// TwinCAT 3 PLC project GettingStarted
// ProgramVersion: 3.1.4026.20
// libraries:
//   Tc2_Standard, * (Beckhoff Automation GmbH)
//   Tc2_System, * (Beckhoff Automation GmbH)
//   Tc2_TcpIp, * (Beckhoff Automation GmbH)
//   Tc2_Utilities, * (Beckhoff Automation GmbH)
//   Tc3_Module, * (Beckhoff Automation GmbH)
// project tree:
//   / PlcTask.TcTTO
//   POUs/ FB_TCPClient.TcPOU, FB_TCPServer.TcPOU, MAIN.TcPOU
// real-time tasks:
//   TASK PlcTask: cycle T#10ms, priority 20, ADS port 350

CONFIGURATION GettingStarted
    RESOURCE PLC ON TwinCAT3
        TASK PlcTask(INTERVAL := T#10ms, PRIORITY := 20);
        PROGRAM MAIN WITH PlcTask : MAIN;
    END_RESOURCE
END_CONFIGURATION

// ---- POUs/MAIN.TcPOU
PROGRAM MAIN
VAR
	bInit: BOOL := TRUE;
	fbSocketCloseAll: FB_SocketCloseAll; 
	bSocketCloseError: BOOL;
	nSocketCloseError: UDINT;
	
	fbTcpClient1					: FB_TCPClient;
		sClient1SendData			: STRING(255);
		nServer1Port				: UDINT 				:= 12000;
		sServer1Host				: T_IPv4Addr 			:= '127.0.0.1';
		bStartClient1Communication	: BOOL 					:= TRUE;
		tClient1CycleTime			: TIME 					:= T#0.5S;
		bClient1SendTrigger			: BOOL;
		bClient1Connected			: BOOL;
		sClient1ReceivedData		: STRING(255);
		bClient1Busy				: BOOL;
		bClientError1				: BOOL;
		nClient1ErrorID1			: UDINT;		
		
	fbTcpEchoServer1				: FB_TCPServer;
		sServerReceivedData			: STRING(255);
		bStartServer1Communication	: BOOL 					:= TRUE;
		bServer1Connected			: BOOL;
		sServerData					: STRING(255);
		bServer1Busy				: BOOL;
		bServer1Error				: BOOL;
		nServer1ErrorID				: UDINT;
	
	bAutogenerateData				: BOOL 					:= TRUE;
	fbTimer1						: TON;
	nCnt							: UDINT;
	
// Optional second Client and Server
(*	fbTcpClient2					: FB_TCPClient;
		sClient2SendData			: STRING(255)			:= 'TestString123';
		sClient2ReceivedData		: STRING(255);			
	fbTcpServer2					: FB_TCPServer;
		sServer2Data				: STRING(255); *)
END_VAR

IF bInit THEN 				// Init Step to close all sockets after login PLC with  downlaod
	fbSocketCloseAll(
		sSrvNetId:= '', 
		bExecute:= TRUE, 
		tTimeout:= T#3S, 
		bBusy=> , 
		bError=> bSocketCloseError, 
		nErrId=> nSocketCloseError);
	IF NOT (fbSocketCloseAll.bBusy OR fbSocketCloseAll.bError) THEN
		bInit := FALSE;
		fbSocketCloseAll(bExecute:= FALSE);
	END_IF
ELSE
	
	fbTcpClient1(
		nRemotePort:= nServer1Port, 								// Server port
		sRemoteHost:= sServer1Host, 								// Server IP (127.0.0.1 for local communication)
		bStartCommunication:= bStartClient1Communication, 			// Start communication, when FALSE, connection is closed
		sSendData:= sClient1SendData, 								// Data that are sent to the server
		tCycleTimeSend:= (*tClient1CycleTime*), 					// TimeInterval for cyclic sending
		bSendTrigger:= ,											// Trigger to send one telegramm manually 
		bConnected => bClient1Connected,							// Switches to TRUE when Client is connected to a server
		sReceivedData=> sClient1ReceivedData,						// Data that are received
		bBusy=> bClient1Busy, 
		bError=> bClientError1, 
		nErrorID=> nClient1ErrorID1, ); 
	
	IF bAutogenerateData AND bClient1Connected THEN
		fbTimer1(IN:= NOT fbTimer1.Q, PT:= tClient1CycleTime, Q=> , ET=> );
		IF fbTimer1.Q  THEN
			sClient1SendData := Concat('TestString No.', UDINT_TO_STRING(nCnt));
			fbTcpClient1.bSendTrigger := TRUE;
			nCnt := nCnt + 1;
		ELSE
			fbTcpClient1.bSendTrigger := FALSE;
		END_IF
	END_IF 
		
	fbTcpEchoServer1(
		sLocalHost:= '0.0.0.0',										// Server IP address to listen on, 0.0.0.0 for listening on all network adapters
		nLocalPort:= nServer1Port, 									// Server port
		bStartCommunication:= bStartServer1Communication, 			// Allow Client-connection or close connection
		bConnected => bServer1Connected,							// Client connection is valid
		sSendData => sServerData,
		bBusy=> bServer1Busy, 
		bError=> bServer1Error, 
		nErrorID=> nServer1ErrorID);
	
	// Optional second Client and Server
	
(*	fbTcpClient2(
		sRemoteHost:= '127.0.0.1', 
		nRemotePort:= 12001, 
		sSendData:= sClient2SendData, 
		bStartCommunication:= TRUE, 
		tCycleTimeSend:= T#2S, 
		bSendTrigger:= ,
		bConnected => , 
		sReceivedData=> sClient2ReceivedData, 
		nErrorID=> , 
		bError=> , 
		bBusy=> );
		
	fbTcpServer2(
		sLocalHost:= '0.0.0.0', 
		nLocalPort:= 12001, 
		bStartCommunication:= TRUE, 
		sSendData => sServer2Data, 
		bBusy=> , 
		bError=> , 
		nErrorID=> ); *)
END_IF

END_PROGRAM

// ---- POUs/FB_TCPClient.TcPOU
FUNCTION_BLOCK FB_TCPClient
VAR_INPUT
	sRemoteHost: T_IPv4Addr;
	nRemotePort: UDINT;
	sSendData: STRING(255);	
	bStartCommunication: BOOL;
	tCycleTimeSend: TIME;
	bSendTrigger : BOOL;
END_VAR
VAR_OUTPUT
	bConnected: BOOL;
	sReceivedData: STRING(255);
	nErrorID: UDINT;
	bError: BOOL;
	bBusy: BOOL;
END_VAR
VAR
	iState: INT;
	fbSocketConnect: FB_SocketConnect;
	fbSocketSend: FB_SocketSend;
	fbSocketClose: FB_SocketClose;
	fbSocketReceive: FB_SocketReceive;
	hSocket: T_HSOCKET;

	fbTimer: TON;
	nRecBytes: UDINT;
	bExecuteSocketSend: BOOL;
	RTrig: R_TRIG;
END_VAR

CASE iState OF
0:	// Init State
	fbSocketConnect(bExecute := FALSE); 
	fbSocketSend(bExecute := FALSE); 
	fbSocketReceive(bExecute := FALSE);
	fbSocketClose(bExecute := FALSE); 
	bConnected := FALSE; 
	bBusy := FALSE;
	IF bStartCommunication = TRUE THEN									// Start communication manually 
		iState := iState + 10;
		bBusy := TRUE;
		bError := FALSE;
	END_IF

10:	// Connect Server
	fbSocketConnect(													// Open connection to server
		sSrvNetId:= '', 
		sRemoteHost:= sRemoteHost, 
		nRemotePort:= nRemotePort, 
		bExecute:= TRUE, 
		tTimeout:= T#4S, 
		bBusy=> , 
		bError=> bError, 
		nErrId=> nErrorID, 
		hSocket=> hSocket);

	IF hSocket.handle <> 0 AND NOT (fbSocketConnect.bBusy) THEN			// Handle is created
		bConnected := TRUE; 
		iState :=iState + 5;
	ELSIF bError THEN
		iState := 0; 	
	END_IF
	
	
15:																		// StartCommunication
	IF (tCycleTimeSend <> T#0MS) THEN									// Send data cyclically
		fbTimer(IN:= NOT fbTimer.Q, PT:= tCycleTimeSend, Q=> , ET=> );		
	END_IF
	RTrig(CLK:= bSendTrigger, Q=> );									// SendData on manuel trigger
	
	fbSocketSend(														// Send Data
		sSrvNetId:= '', 
		hSocket:= hSocket, 
		cbLen:= LEN2(ADR(sSendData)), 
		pSrc:= ADR(sSendData), 
		bExecute:= (fbTimer.Q OR RTrig.Q), 
		tTimeout:= T#2S, 
		bError=> bError, 
		nErrId=> nErrorID, 
		nErrId=> );

	fbSocketReceive(													// ReceiveData
		sSrvNetId:= '', 
		hSocket:= hSocket, 
		cbLen:= SIZEOF(sReceivedData), 
		pDest:=  ADR(sReceivedData), 
		bExecute:= true, 
		tTimeout:= T#3S, 
		bBusy=> , 
		bError=> bError, 
		nErrId=> nErrorID, 
		nRecBytes=> nRecBytes);
		
	IF NOT fbSocketReceive.bBusy THEN									// Check cyclically for new data
		fbSocketReceive(bExecute := FALSE);
	END_IF						
	IF NOT bStartCommunication OR bError THEN							// Close connection in case of error or manual communication stop
		iState := 20;
	END_IF
20: 
	fbSocketClose(														// Close connection
		sSrvNetId:= '', 
		hSocket:= hSocket, 
		bExecute:= TRUE, 
		tTimeout:= T#4S, 
		bBusy=> , 
		bError=> bError, 
		nErrId=> nErrorID );
	IF NOT fbSocketClose.bBusy THEN
		iState :=0;		
	END_IF
END_CASE

END_FUNCTION_BLOCK

// ---- POUs/FB_TCPServer.TcPOU
FUNCTION_BLOCK FB_TCPServer
VAR_INPUT
	sLocalHost: T_IPv4Addr;
	nLocalPort: UDINT;
	bStartCommunication : BOOL;
END_VAR
VAR_OUTPUT
	bConnected: BOOL;
	sSendData: STRING(255);
	bBusy: BOOL;	
	bError: BOOL;
	nErrorID: UDINT;
END_VAR
VAR
	iState: INT;
	hListener: T_HSOCKET;
	hSocket: T_HSOCKET;
	fbSocketAccept: FB_SocketAccept;
	fbSocketListen: FB_SocketListen;
	fbSocketReceive: FB_SocketReceive;
	fbSocketClose: FB_SocketClose;
	fbSocketCloseAll: FB_SocketCloseAll;
	fbSocketSend: FB_SocketSend;
	bAcceptExecute: BOOL;
	
	ReceiveCounter: UDINT;
	sReadData: STRING(255);
	
	bSendTrigger: BOOL;
END_VAR

CASE iState OF
0: // Init State
	IF bStartCommunication = TRUE  THEN
		fbSocketListen(bExecute := FALSE);
		fbSocketAccept(bExecute := FALSE);
		fbSocketCloseAll(bExecute := FALSE);
		fbSocketClose(bExecute:= FALSE);
		bBusy := TRUE;
		iState := iState + 10;
	ELSE
		bBusy := FALSE;
	END_IF
	
10:
	fbSocketListen(																// Open Listener-Socket
		sSrvNetId:= '', 														// Local NetID
		sLocalHost:= sLocalHost, 												// Local IP
		nLocalPort:= nLocalPort, 												// Local Port
		bExecute:= TRUE, 
		tTimeout:= T#4S, 
		bBusy=> , 
		bError=> bError, 
		nErrId=> nErrorID,
		hListener=> hListener);													// Handle of Listener Socket
		
	IF hListener.handle <> 0 THEN
		iState := iState + 10;	
	ELSIF bError THEN
		iState := 40;
	END_IF
	
20: 		
	fbSocketAccept(																// Accept Client connection
		sSrvNetId:= '', 		
		hListener:= hListener, 													// Handle of Listener Socket
		bExecute:= TRUE, 
		tTimeout:= T#4S, 
		bAccepted=> , 
		bBusy=> , 
		bError=> bError, 
		nErrId=> nErrorID,
		hSocket=> hSocket);														// Connection Handle
	IF NOT fbSocketAccept.bBusy THEN
		fbSocketAccept(bExecute:= FALSE);
	END_IF

	IF bError THEN
		iState := 40; 
	ELSIF hSocket.handle <> 0 THEN
		iState := iState + 10; 
		bConnected := TRUE;
	END_IF
	
30: // Receive Data
	fbSocketReceive(															// Check cyclically for new client telegrams 
		sSrvNetId:= '', 
		hSocket:= hSocket, 
		cbLen:= SIZEOF(sReadData) , 
		pDest:= ADR(sReadData), 
		bExecute:= TRUE, 														
		tTimeout:= T#4S, 
		bBusy=> , 
		bError=> bError, 
		nErrId=> nErrorID,
		nRecBytes=> );
		
	IF NOT fbSocketReceive.bBusy THEN
		fbSocketReceive(bExecute := FALSE);
		IF fbSocketReceive.nRecBytes <> 0 THEN									// Switch to send-state when data are received
			fbSocketSend(bExecute:= FALSE);
			ReceiveCounter := ReceiveCounter + 1; 
			memcpy(ADR(sSendData), ADR(sReadData), fbSocketReceive.nRecBytes);	// Copy received data from ReceiveBuffer to SendBuffer
			memset(ADR(sReadData), 0, SIZEOF(sReadData));						// Empty ReceiveBuffer
			iState := iState + 5;
		END_IF
	END_IF
	IF fbSocketReceive.bError OR(NOT bStartCommunication) THEN					// Close connection when error is occuring or trigger is set
		iState := iState + 10;
	END_IF

35: // Send Data
	fbSocketSend(																// Send Data to client
		sSrvNetId:= '', 
		hSocket:= hSocket, 
		cbLen:= LEN2(ADR(sSendData)), 
		pSrc:= ADR(sSendData),
		bExecute:= TRUE, 
		tTimeout:= T#3S, 
		bBusy=> , 
		bError=> bError, 
		nErrId=> nErrorID);	
	
	
	IF NOT fbSocketSend.bBusy THEN												// Switch back to receiving state after sending
		iState := iState - 5;
	ELSIF fbSocketSend.bError THEN
		iState := iState + 5;													// Close connection in case of error 
	END_IF
	
40:	// Error Handling	
	fbSocketClose(																// Close Listener-Socket
		sSrvNetId:= '', 
		hSocket:= hListener, 
		bExecute:= TRUE, 
		tTimeout:= T#4S, 
		bBusy=> , 
		bError=> bError, 
		nErrId=> nErrorID);		
	IF (NOT fbSocketClose.bBusy) OR fbSocketClose.bError THEN
		hListener.handle := 0;
		iState := iState + 1;
	END_IF
41:	
	fbSocketClose(bExecute := FALSE);
	iState := iState + 1;
42:
	fbSocketClose(																// Close Connection Socket
		sSrvNetId:= '', 
		hSocket:= hSocket, 
		bExecute:= TRUE, 
		tTimeout:= T#4S, 
		bBusy=> , 
		bError=> bError, 
		nErrId=> nErrorID);
	IF NOT (fbSocketClose.bBusy) OR fbSocketClose.bError THEN
		hSocket.handle := 0;	
		iState := 0;
		bConnected := FALSE;
	END_IF
END_CASE

END_FUNCTION_BLOCK
